Fanuc KAREL source: kt00337.KL

-- PROVISIONAL review KL for V1013-1; original PC SHA256 8fe7e45802a31b145a6951a8c2e4d42c8927833f51b322b5aaa0032ae0445153
-- Incomplete behavior may be omitted. Consult companion uncertainty JSON. Do not deploy.
PROGRAM KT00337
%NOLOCKGROUP
VAR
  B1 : BOOLEAN
  B2 : BOOLEAN
  OUT : BOOLEAN
BEGIN
  -- UNRESOLVED_PC offsets 5-12; opcodes 9D,23
  -- UNRESOLVED_PC offsets 17-24; opcodes 9C,23
  -- UNRESOLVED_PC offsets 29-36; opcodes 9D,23
  -- UNRESOLVED_PC offsets 41-48; opcodes 9C,23
  -- UNRESOLVED_PC offsets 53-72; opcodes 21,21,59,23
  -- UNRESOLVED_PC offsets 77-81; opcodes 7F
END KT00337
